(*
A circular queue implementation for managing `I_Arg`.  
*)
FUNCTION_BLOCK ArgQueue
VAR_GENERIC CONSTANT
	nCap		: UDINT := 100;
END_VAR

IMPLEMENTS I_MutArgQueue

VAR
	_list		: ArgList<nCap>;
	_nLen		: UDINT := 0;
	_nHead		: UDINT := 1;
	_nTail		: UDINT := 1;
END_VAR

(*
Clears the queue.
*)
METHOD Clear
_nHead := 1;
_nTail := 1;
_nLen := 0;
_list.Set(0, 1);
END_METHOD

(*
Returns the current head index of the queue, indicating the next position for insertion.
*)
PROPERTY Head : UDINT
GET
Head := _nHead;
END_GET
END_PROPERTY

PROPERTY Length : UDINT
GET
Length := _nLen;
END_GET
END_PROPERTY

(*
Provides access to the underlying list structure that holds the queue's argument objects.
*)
PROPERTY List : I_ArgList
GET
List := _list;
END_GET
END_PROPERTY

(*
Allows initializing an external interface variable with an interface pointer to this instance within declaration block.
Example:
iQueue: I_MutArgQueue;
queue: ArgQueue := (MutProxy := iQueue);
Result: iQueue <> 0 
*)
PROPERTY MutProxy : REFERENCE TO I_MutArgQueue
SET
MutProxy := THIS^;
END_SET
END_PROPERTY

(*
Retrieves and removes the next argument from the queue.  
Advances the tail pointer, ensuring cyclic operation within the queue's capacity.
Returns:
- Ok - Returns `I_Arg`.
- Err.NotFound - Returns null, queue empty.
- Check `I_ArgList.Get` for more results.
*)
METHOD Pop : Result
VAR_INPUT
	iOut	: REFERENCE TO I_Arg;
END_VAR
IF _nLen = 0 THEN
	Pop := Err.NotFound;
	RETURN;
END_IF;

IF IsOk(_list.Get(_nHead, iOut), nOut => Pop) THEN
	_nHead := (_nHead MOD nCap) + 1;
	_nLen := _nLen - 1;
	Pop := Ok;
END_IF;
END_METHOD

(*
Allows initializing an external interface variable with an interface pointer to this instance within declaration block.
Example:
iQueue: I_ArgQueue;
queue: ArgQueue := (Proxy := iQueue);
Result: iQueue <> 0 
*)
PROPERTY Proxy : REFERENCE TO I_ArgQueue
SET
Proxy := THIS^;
END_SET
END_PROPERTY

(*
Adds a new argument to the queue.  
Advances the head pointer while maintaining a cyclic structure, and returns an overflow error if the queue is full.
Returns:
- Ok - Successful insertion
- Err.Ovf - Returns null, the queue is full.
- Check `I_ArgList.Set` for more results.
*)
METHOD Push : Result
VAR_INPUT
	iIn		: I_Arg;
END_VAR
IF _nLen = nCap THEN
	Push := Err.Ovf;
	RETURN;
END_IF;

IF IsOk(_list.Set(iIn, _nTail), nOut => Push) THEN
	_nTail := (_nTail MOD nCap) + 1;
	_nLen := _nLen + 1;
	Push := Ok;
END_IF;
END_METHOD

(*
Returns the current tail index of the queue, indicating the next position for retrieval.
*)
PROPERTY Tail : UDINT
GET
Tail := _nTail;
END_GET
END_PROPERTY

END_FUNCTION_BLOCK

(* stored: Version 1.1.0.1
   POU ArgQueue: Id {c76e1546-2227-4293-8d71-24ba2b1f9980}, SpecialFunc None
   Folder Proxy: Id {9f39ca87-734b-4ce2-a064-6cb3a1e15ca4}
   Method Clear: Id {de26b2be-362d-4495-b24f-d07023138547}
   Property Head: Id {c9aced8c-5615-4602-a8c9-d2cca06beb56}
   Get Get: Id {e1f4e3bb-f456-4b54-a664-6226a1648088}
   Property Length: Id {138194cb-0617-4188-9db7-14d43055e764}
   Get Get: Id {c65e8145-303d-4803-99d0-e1f5bad90830}
   Property List: Id {cf73eedb-24ba-4099-8ac4-bd0f99e7e007}
   Get Get: Id {fcb1b69f-2ae2-4e8b-8036-3051766ec0a1}
   Property MutProxy: Id {df8ba48c-7672-4a55-b0be-3b5f9a4d9dff}
   Set Set: Id {e645097b-951f-44f1-9c61-03dc6b075533}
   Method Pop: Id {ebbd8206-4440-4673-b31a-c80b5ef2f1c1}
   Property Proxy: Id {0a9d7853-91a6-46b9-8229-824366fef474}
   Set Set: Id {3ef5d859-90d8-4433-81d3-8c4a83e9ef75}
   Method Push: Id {7a6a861d-ce7d-4b8e-83b1-463d9bd37168}
   Property Tail: Id {86561c9d-d0a1-4b85-b773-d6ff1230d5fb}
   Get Get: Id {97904e90-29ab-41d0-962b-7b170142aeb0} *)
